# EPICS autosave request: iocs/kinetixIOC/iocBoot/iocKinetix/auto_settings.req
file "ADKinetix_settings.req",      P=$(P),  R=cam1:
file "NDStdArrays_settings.req",    P=$(P),  R=image:
file "commonPlugin_settings.req",   P=$(P)
